(* Logix 5000 project; controller Google vendor 1 type 14 code 151 rev 31.11; software revision 31.00 *)

TASK MainTask (continuous, watchdog 500 ms) : MainProgram

MODULES
   Local : vendor 1 type 14 code 151 (Compact 0, rev 31.11)
      Discrete_IO : Embedded (Compact 1, rev 3.1, Output RPI 20 ms)
      Analog_IO : Embedded (Compact 2, rev 1.1, Output RPI 80 ms)
      Counters : Embedded (Compact 3, rev 1.1, Output RPI 20 ms)
      Lift_Main_Drive : PowerFlex 525-EENET (Ethernet 192.168.1.42, rev 5.1, Output RPI 50 ms)
      LST_1 : vendor 678 type 100 code 276 (Ethernet 192.168.1.149, rev 11.1, Output RPI 19 ms)
      LST_2 : vendor 678 type 100 code 276 (Ethernet 192.168.1.50, rev 11.1, Output RPI 17 ms)
      ToteCodeReader : vendor 678 type 773 code 1307 (Ethernet 192.168.1.151, rev 1.1, Output RPI 60 ms)
      L5_Conv : vendor 629 type 43 code 2 (Ethernet 192.168.1.165, rev 2.1, StandardDataDriven RPI 30 ms)
      L4_Conv : vendor 629 type 43 code 2 (Ethernet 192.168.1.164, rev 2.1, StandardDataDriven RPI 30 ms)
      L1_Conv : vendor 629 type 43 code 2 (Ethernet 192.168.1.161, rev 2.1, StandardDataDriven RPI 30 ms)
      Infeed_Conv : vendor 629 type 43 code 2 (Ethernet 192.168.1.160, rev 2.1, StandardDataDriven RPI 30 ms)
           Infeed_Conv:I.Data[0].0   // Zone 1 Sensor
           Infeed_Conv:I.Data[0].1   // Zone 2 Sensor
           Infeed_Conv:I.Data[0].2   // Zone 3 Sensor
           Infeed_Conv:I.Data[0].3   // Zone 4 Sensor
      L2_Conv : vendor 629 type 43 code 2 (Ethernet 192.168.1.162, rev 2.1, StandardDataDriven RPI 30 ms)
      L3_Conv : vendor 629 type 43 code 2 (Ethernet 192.168.1.163, rev 2.1, StandardDataDriven RPI 30 ms)
      Lift_Conv : vendor 629 type 43 code 2 (Ethernet 192.168.1.166, rev 2.1, StandardDataDriven RPI 30 ms)
END_MODULES

TYPE Addr :   // Structure UDT for MSG UDT
STRUCT
   Family : INT;   // 2 for IP4
   Port : INT;   // Remote Port Number
   Addr : DINT;   // Remote IP Address
END_STRUCT
END_TYPE

TYPE GIB_MSG :   // UDT Specified by Rockwell
STRUCT
   Instance : DINT;
   Addr : Addr;
END_STRUCT
END_TYPE

TYPE State :
STRUCT
   Stopped : DINT;
   Resetting : DINT;
   Ready : DINT;
   Starting : DINT;
   Running : DINT;
   Stopping : DINT;
END_STRUCT
END_TYPE

ADD_ON_INSTRUCTION Conv_Sensor_Inputs   (* revision 1.0 *)
VAR_INPUT
   Data : SINT; {required}
END_VAR
VAR_OUTPUT
   Input_0 : BOOL; {access Read Only, required}
   Input_1 : BOOL; {access Read Only, required}
   Input_2 : BOOL; {access Read Only, required}
   Input_3 : BOOL; {access Read Only, required}
END_VAR
VAR_INPUT
   Infeed_Mode : BOOL; {required}
   Outfeed_Mode : BOOL; {required}
   Outfeed_Stop_Delay : DINT; {required}
END_VAR
VAR
   Input_Delay : TIMER[4] := ([0].PRE := 1000, [1].PRE := 1000, [2].PRE := 1000, [3].PRE := 1000); {access None}
END_VAR

ROUTINE Logic   (* ladder *)
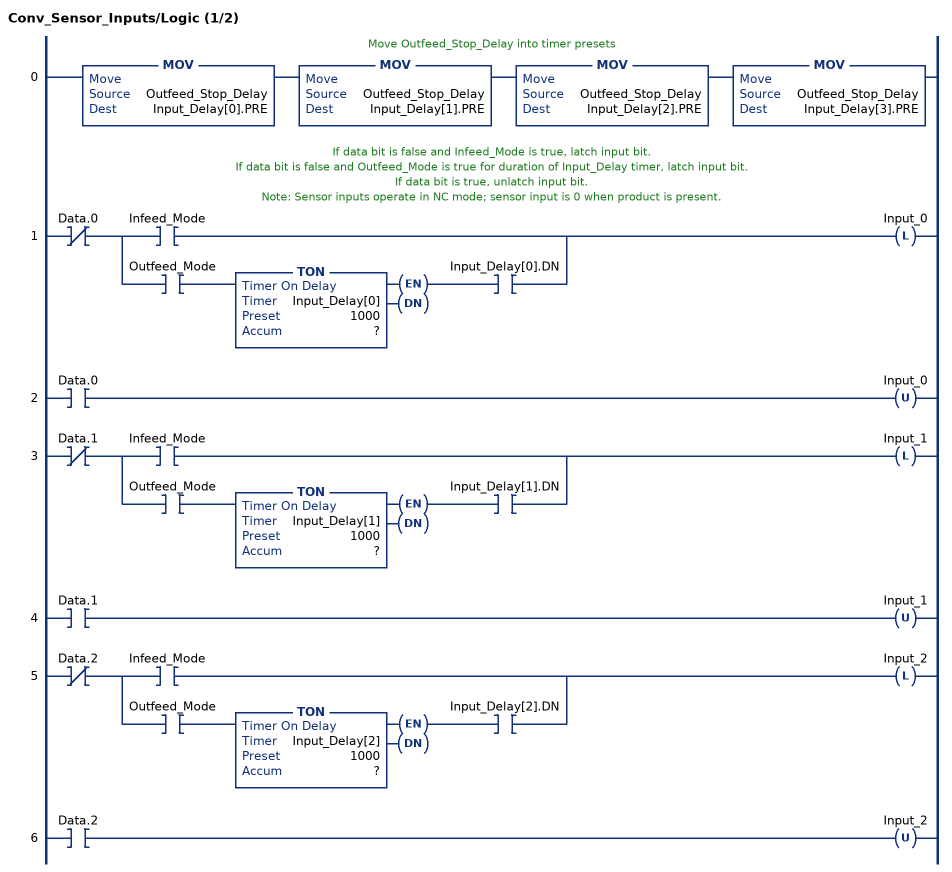
   // Move Outfeed_Stop_Delay into timer presets
   0: MOV(Outfeed_Stop_Delay,Input_Delay[0].PRE)MOV(Outfeed_Stop_Delay,Input_Delay[1].PRE)MOV(Outfeed_Stop_Delay,Input_Delay[2].PRE)MOV(Outfeed_Stop_Delay,Input_Delay[3].PRE);
   // If data bit is false and Infeed_Mode is true, latch input bit.
   // If data bit is false and Outfeed_Mode is true for duration of Input_Delay timer, latch input bit.
   // If data bit is true, unlatch input bit.
   // Note: Sensor inputs operate in NC mode; sensor input is 0 when product is present.
   1: XIO(Data.0)[XIC(Infeed_Mode) ,XIC(Outfeed_Mode) TON(Input_Delay[0],?,?) XIC(Input_Delay[0].DN) ]OTL(Input_0);
   2: XIC(Data.0)OTU(Input_0);
   3: XIO(Data.1)[XIC(Infeed_Mode) ,XIC(Outfeed_Mode) TON(Input_Delay[1],?,?) XIC(Input_Delay[1].DN) ]OTL(Input_1);
   4: XIC(Data.1)OTU(Input_1);
   5: XIO(Data.2)[XIC(Infeed_Mode) ,XIC(Outfeed_Mode) TON(Input_Delay[2],?,?) XIC(Input_Delay[2].DN) ]OTL(Input_2);
   6: XIC(Data.2)OTU(Input_2);
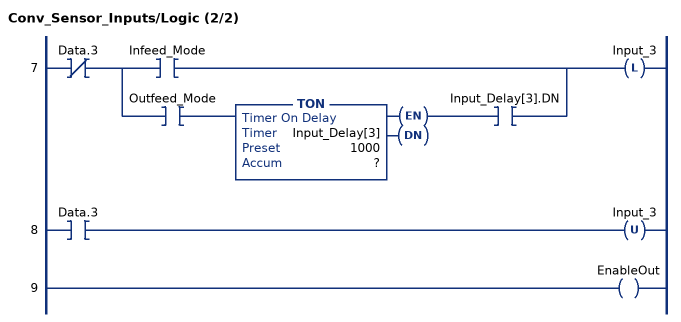
   7: XIO(Data.3)[XIC(Infeed_Mode) ,XIC(Outfeed_Mode) TON(Input_Delay[3],?,?) XIC(Input_Delay[3].DN) ]OTL(Input_3);
   8: XIC(Data.3)OTU(Input_3);
   9: OTE(EnableOut);
END_ROUTINE
END_ADD_ON_INSTRUCTION

ADD_ON_INSTRUCTION Conveyor_Motor_Control   (* revision 1.0 *)
VAR_OUTPUT
   Motor1_Data : SINT; {required}
   Motor2_Data : SINT; {access Read Only, required}
   Motor3_Data : SINT; {access Read Only, required}
   Motor4_Data : SINT; {access Read Only, required}
END_VAR
VAR_INPUT
   Motor1_FWD : BOOL; {required}
   Motor1_REV : BOOL; {required}
   Motor2_FWD : BOOL; {required}
   Motor2_REV : BOOL; {required}
   Motor3_FWD : BOOL; {required}
   Motor3_REV : BOOL; {required}
   Motor4_FWD : BOOL; {required}
   Motor4_REV : BOOL; {required}
   FWD_Speed : DINT; {required}
   REV_Speed : DINT; {required}
   Start_Delay : DINT; {required}
   Run_Permissive : DINT; {required}
END_VAR
VAR
   FWD_Delay : TIMER[4] := ([0].PRE := 500, [1].PRE := 500, [2].PRE := 500, [3].PRE := 500); {access None}
   REV_Delay : TIMER[4] := ([0].PRE := 500, [1].PRE := 500, [2].PRE := 500, [3].PRE := 500); {access None}
END_VAR

ROUTINE Logic   (* ladder *)
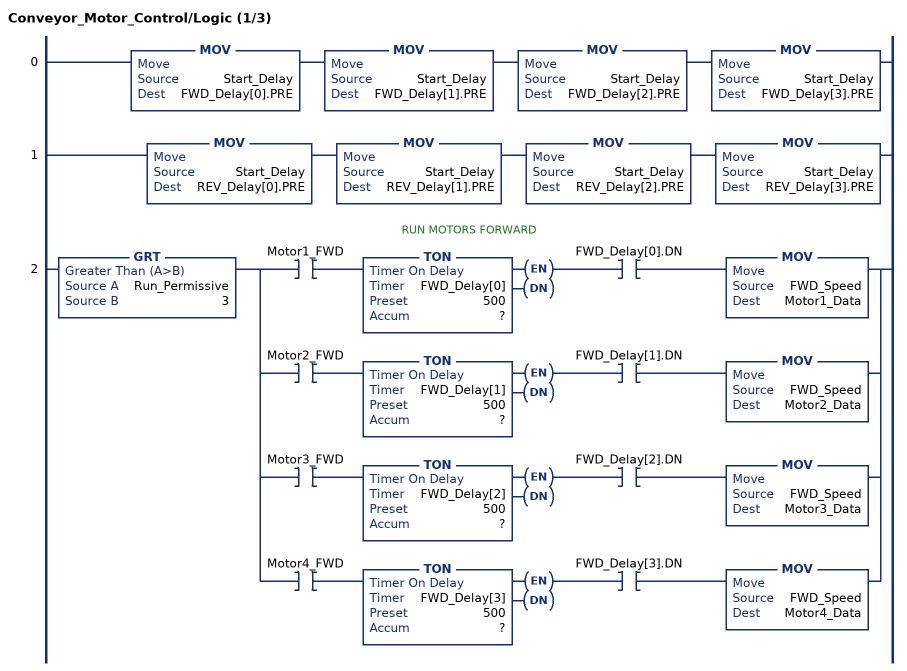
   0: MOV(Start_Delay,FWD_Delay[0].PRE)MOV(Start_Delay,FWD_Delay[1].PRE)MOV(Start_Delay,FWD_Delay[2].PRE)MOV(Start_Delay,FWD_Delay[3].PRE);
   1: MOV(Start_Delay,REV_Delay[0].PRE)MOV(Start_Delay,REV_Delay[1].PRE)MOV(Start_Delay,REV_Delay[2].PRE)MOV(Start_Delay,REV_Delay[3].PRE);
   // RUN MOTORS FORWARD
   2: GRT(Run_Permissive,3)[XIC(Motor1_FWD) TON(FWD_Delay[0],?,?) XIC(FWD_Delay[0].DN) MOV(FWD_Speed,Motor1_Data) ,XIC(Motor2_FWD) TON(FWD_Delay[1],?,?) XIC(FWD_Delay[1].DN) MOV(FWD_Speed,Motor2_Data) ,XIC(Motor3_FWD) TON(FWD_Delay[2],?,?) XIC(FWD_Delay[2].DN) MOV(FWD_Speed,Motor3_Data) ,XIC(Motor4_FWD) TON(FWD_Delay[3],?,?) XIC(FWD_Delay[3].DN) MOV(FWD_Speed,Motor4_Data) ];
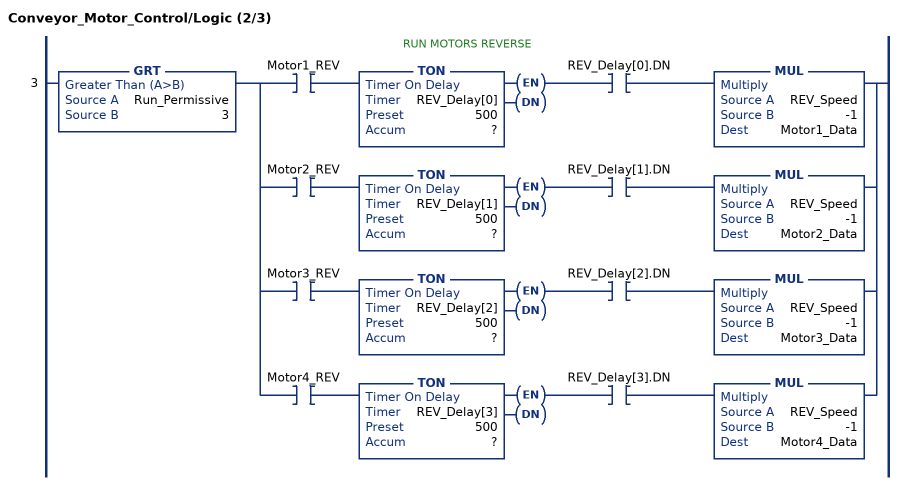
   // RUN MOTORS REVERSE
   3: GRT(Run_Permissive,3)[XIC(Motor1_REV) TON(REV_Delay[0],?,?) XIC(REV_Delay[0].DN) MUL(REV_Speed,-1,Motor1_Data) ,XIC(Motor2_REV) TON(REV_Delay[1],?,?) XIC(REV_Delay[1].DN) MUL(REV_Speed,-1,Motor2_Data) ,XIC(Motor3_REV) TON(REV_Delay[2],?,?) XIC(REV_Delay[2].DN) MUL(REV_Speed,-1,Motor3_Data) ,XIC(Motor4_REV) TON(REV_Delay[3],?,?) XIC(REV_Delay[3].DN) MUL(REV_Speed,-1,Motor4_Data) ];
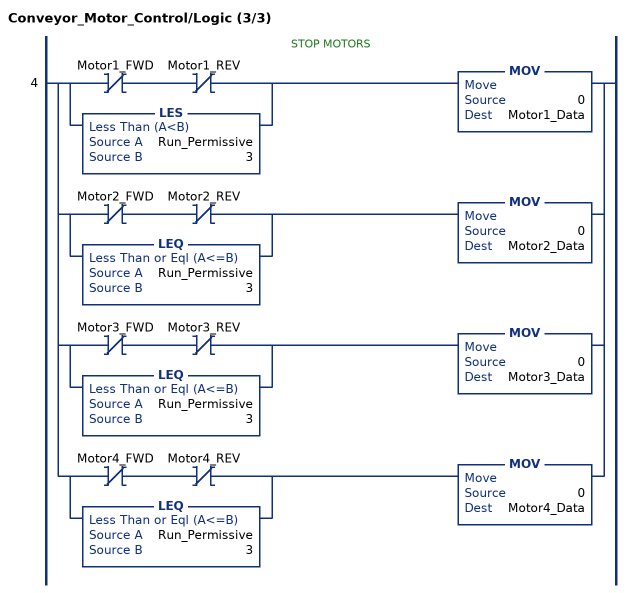
   // STOP MOTORS
   4: [[XIO(Motor1_FWD) XIO(Motor1_REV) ,LES(Run_Permissive,3) ] MOV(0,Motor1_Data) ,[XIO(Motor2_FWD) XIO(Motor2_REV) ,LEQ(Run_Permissive,3) ] MOV(0,Motor2_Data) ,[XIO(Motor3_FWD) XIO(Motor3_REV) ,LEQ(Run_Permissive,3) ] MOV(0,Motor3_Data) ,[XIO(Motor4_FWD) XIO(Motor4_REV) ,LEQ(Run_Permissive,3) ] MOV(0,Motor4_Data) ];
END_ROUTINE
END_ADD_ON_INSTRUCTION

ADD_ON_INSTRUCTION End_Zone_Data   (* revision 1.0 *)
VAR_IN_OUT
   Product_Name : STRING; {required}
   Product_Code : DINT; {required}
END_VAR
VAR_OUTPUT
   Occupied : BOOL; {access Read Only, visible}
END_VAR
VAR_INPUT
   Input : BOOL; {required}
END_VAR
VAR_IN_OUT
   Upstream_ProdName : STRING; {required}
   Upstream_ProdCode : DINT; {required}
END_VAR
VAR_INPUT
   FWD_Direction : BOOL; {required}
   REV_Direction : BOOL; {required}
END_VAR
VAR
   Blank_String : STRING; {access None}
   ONS : DINT; {access None}
   Occupied_Delay : TIMER := (PRE := 20); {access None}
END_VAR

ROUTINE Logic   (* ladder *)
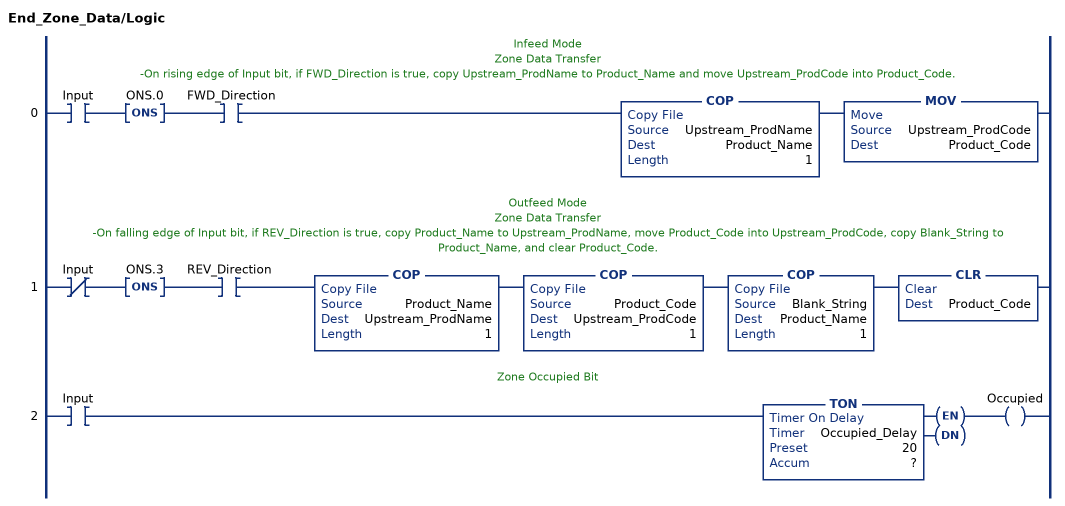
   // Infeed Mode
   // Zone Data Transfer
   // -On rising edge of Input bit, if FWD_Direction is true, copy Upstream_ProdName to Product_Name and move Upstream_ProdCode into Product_Code.
   0: XIC(Input)ONS(ONS.0)XIC(FWD_Direction)COP(Upstream_ProdName,Product_Name,1)MOV(Upstream_ProdCode,Product_Code);
   // Outfeed Mode
   // Zone Data Transfer
   // -On falling edge of Input bit, if REV_Direction is true, copy Product_Name to Upstream_ProdName, move Product_Code into Upstream_ProdCode, copy Blank_String to Product_Name, and clear Product_Code.
   1: XIO(Input)ONS(ONS.3)XIC(REV_Direction)COP(Product_Name,Upstream_ProdName,1)COP(Product_Code,Upstream_ProdCode,1)COP(Blank_String,Product_Name,1)CLR(Product_Code);
   // Zone Occupied Bit
   2: XIC(Input)TON(Occupied_Delay,?,?)OTE(Occupied);
END_ROUTINE
END_ADD_ON_INSTRUCTION

ADD_ON_INSTRUCTION Input_16_Bit   (* revision 1.0 *)
VAR_INPUT
   Data : INT; {required}
END_VAR
VAR_OUTPUT
   Input_0 : BOOL; {access Read Only, required}
END_VAR
VAR_INPUT
   Input0_On_Debounce : DINT; {required}
   Input0_Off_Debounce : DINT; {required}
END_VAR
VAR_OUTPUT
   Input_1 : BOOL; {access Read Only, required}
END_VAR
VAR_INPUT
   Input1_On_Debounce : DINT; {required}
   Input1_Off_Debounce : DINT; {required}
END_VAR
VAR_OUTPUT
   Input_2 : BOOL; {access Read Only, required}
END_VAR
VAR_INPUT
   Input2_On_Debounce : DINT; {required}
   Input2_Off_Debounce : DINT; {required}
END_VAR
VAR_OUTPUT
   Input_3 : BOOL; {access Read Only, required}
END_VAR
VAR_INPUT
   Input3_On_Debounce : DINT; {required}
   Input3_Off_Debounce : DINT; {required}
END_VAR
VAR_OUTPUT
   Input_4 : BOOL; {access Read Only, required}
END_VAR
VAR_INPUT
   Input4_On_Debounce : DINT; {required}
   Input4_Off_Debounce : DINT; {required}
END_VAR
VAR_OUTPUT
   Input_5 : BOOL; {access Read Only, required}
END_VAR
VAR_INPUT
   Input5_On_Debounce : DINT; {required}
   Input5_Off_Debounce : DINT; {required}
END_VAR
VAR_OUTPUT
   Input_6 : BOOL; {access Read Only, required}
END_VAR
VAR_INPUT
   Input6_On_Debounce : DINT; {required}
   Input6_Off_Debounce : DINT; {required}
END_VAR
VAR_OUTPUT
   Input_7 : BOOL; {access Read Only, required}
END_VAR
VAR_INPUT
   Input7_On_Debounce : DINT; {required}
   Input7_Off_Debounce : DINT; {required}
END_VAR
VAR_OUTPUT
   Input_8 : BOOL; {access Read Only, required}
END_VAR
VAR_INPUT
   Input8_On_Debounce : DINT; {required}
   Input8_Off_Debounce : DINT; {required}
END_VAR
VAR_OUTPUT
   Input_9 : BOOL; {access Read Only, required}
END_VAR
VAR_INPUT
   Input9_On_Debounce : DINT; {required}
   Input9_Off_Debounce : DINT; {required}
END_VAR
VAR_OUTPUT
   Input_10 : BOOL; {access Read Only, required}
END_VAR
VAR_INPUT
   Input10_On_Debounce : DINT; {required}
   Input10_Off_Debounce : DINT; {required}
END_VAR
VAR_OUTPUT
   Input_11 : BOOL; {access Read Only, required}
END_VAR
VAR_INPUT
   Input11_On_Debounce : DINT; {required}
   Input11_Off_Debounce : DINT; {required}
END_VAR
VAR_OUTPUT
   Input_12 : BOOL; {access Read Only, required}
END_VAR
VAR_INPUT
   Input12_On_Debounce : DINT; {required}
   Input12_Off_Debounce : DINT; {required}
END_VAR
VAR_OUTPUT
   Input_13 : BOOL; {access Read Only, required}
END_VAR
VAR_INPUT
   Input13_On_Debounce : DINT; {required}
   Input13_Off_Debounce : DINT; {required}
END_VAR
VAR_OUTPUT
   Input_14 : BOOL; {access Read Only, required}
END_VAR
VAR_INPUT
   Input14_On_Debounce : DINT; {required}
   Input14_Off_Debounce : DINT; {required}
END_VAR
VAR_OUTPUT
   Input_15 : BOOL; {access Read Only, required}
END_VAR
VAR_INPUT
   Input15_On_Debounce : DINT; {required}
   Input15_Off_Debounce : DINT; {required}
END_VAR
VAR
   Debounce_On_TMR : TIMER[16]; {access None}
   Debounce_Off_TMR : TIMER[16]; {access None}
END_VAR

ROUTINE Logic   (* ladder *)
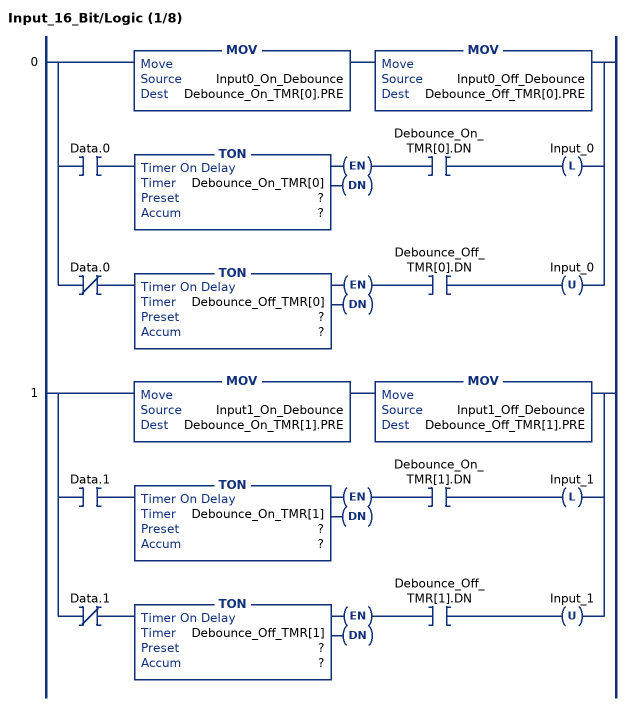
   0: [MOV(Input0_On_Debounce,Debounce_On_TMR[0].PRE) MOV(Input0_Off_Debounce,Debounce_Off_TMR[0].PRE) ,[XIC(Data.0) TON(Debounce_On_TMR[0],?,?) XIC(Debounce_On_TMR[0].DN) OTL(Input_0) ,XIO(Data.0) TON(Debounce_Off_TMR[0],?,?) XIC(Debounce_Off_TMR[0].DN) OTU(Input_0) ] ];
   1: [MOV(Input1_On_Debounce,Debounce_On_TMR[1].PRE) MOV(Input1_Off_Debounce,Debounce_Off_TMR[1].PRE) ,[XIC(Data.1) TON(Debounce_On_TMR[1],?,?) XIC(Debounce_On_TMR[1].DN) OTL(Input_1) ,XIO(Data.1) TON(Debounce_Off_TMR[1],?,?) XIC(Debounce_Off_TMR[1].DN) OTU(Input_1) ] ];
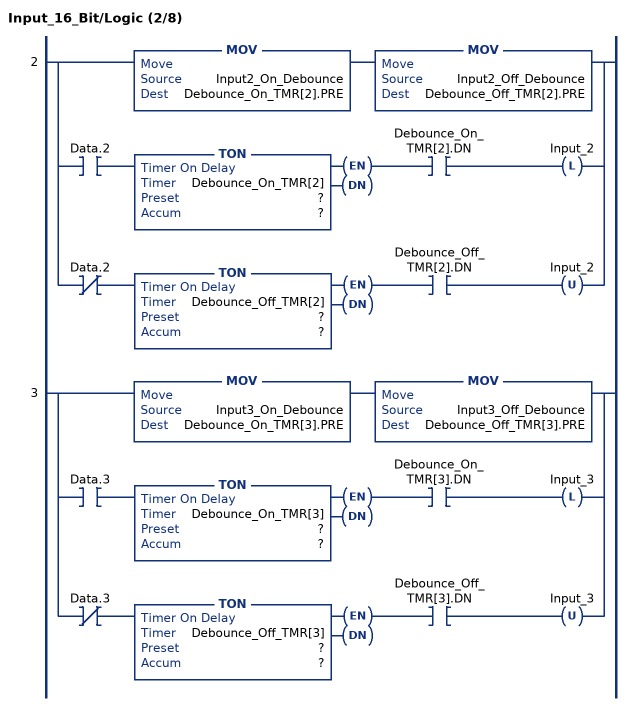
   2: [MOV(Input2_On_Debounce,Debounce_On_TMR[2].PRE) MOV(Input2_Off_Debounce,Debounce_Off_TMR[2].PRE) ,[XIC(Data.2) TON(Debounce_On_TMR[2],?,?) XIC(Debounce_On_TMR[2].DN) OTL(Input_2) ,XIO(Data.2) TON(Debounce_Off_TMR[2],?,?) XIC(Debounce_Off_TMR[2].DN) OTU(Input_2) ] ];
   3: [MOV(Input3_On_Debounce,Debounce_On_TMR[3].PRE) MOV(Input3_Off_Debounce,Debounce_Off_TMR[3].PRE) ,[XIC(Data.3) TON(Debounce_On_TMR[3],?,?) XIC(Debounce_On_TMR[3].DN) OTL(Input_3) ,XIO(Data.3) TON(Debounce_Off_TMR[3],?,?) XIC(Debounce_Off_TMR[3].DN) OTU(Input_3) ] ];
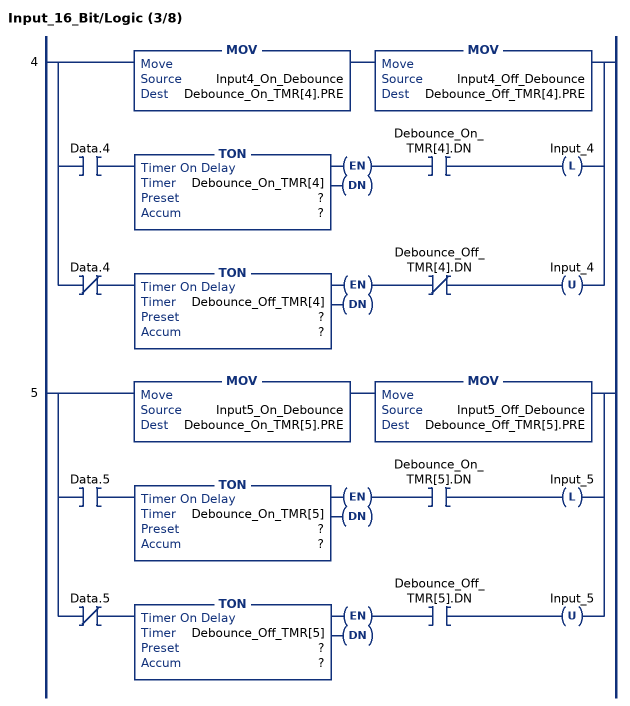
   4: [MOV(Input4_On_Debounce,Debounce_On_TMR[4].PRE) MOV(Input4_Off_Debounce,Debounce_Off_TMR[4].PRE) ,[XIC(Data.4) TON(Debounce_On_TMR[4],?,?) XIC(Debounce_On_TMR[4].DN) OTL(Input_4) ,XIO(Data.4) TON(Debounce_Off_TMR[4],?,?) XIO(Debounce_Off_TMR[4].DN) OTU(Input_4) ] ];
   5: [MOV(Input5_On_Debounce,Debounce_On_TMR[5].PRE) MOV(Input5_Off_Debounce,Debounce_Off_TMR[5].PRE) ,[XIC(Data.5) TON(Debounce_On_TMR[5],?,?) XIC(Debounce_On_TMR[5].DN) OTL(Input_5) ,XIO(Data.5) TON(Debounce_Off_TMR[5],?,?) XIC(Debounce_Off_TMR[5].DN) OTU(Input_5) ] ];
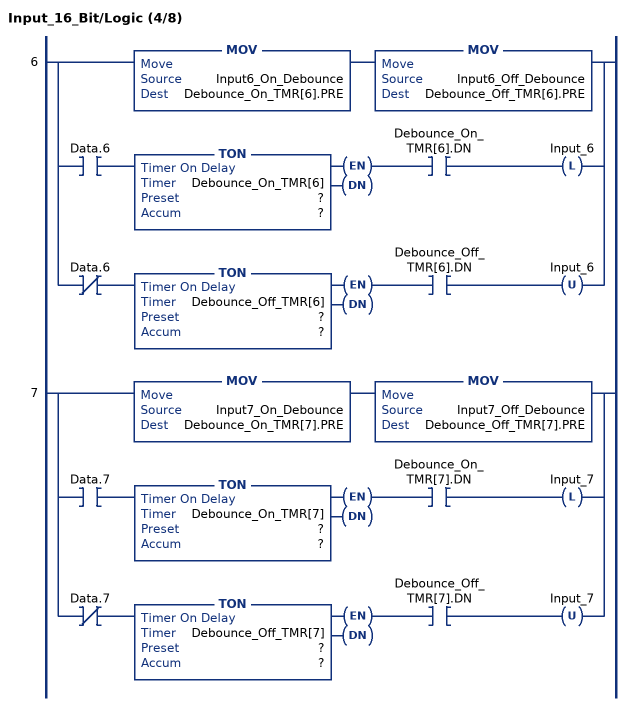
   6: [MOV(Input6_On_Debounce,Debounce_On_TMR[6].PRE) MOV(Input6_Off_Debounce,Debounce_Off_TMR[6].PRE) ,[XIC(Data.6) TON(Debounce_On_TMR[6],?,?) XIC(Debounce_On_TMR[6].DN) OTL(Input_6) ,XIO(Data.6) TON(Debounce_Off_TMR[6],?,?) XIC(Debounce_Off_TMR[6].DN) OTU(Input_6) ] ];
   7: [MOV(Input7_On_Debounce,Debounce_On_TMR[7].PRE) MOV(Input7_Off_Debounce,Debounce_Off_TMR[7].PRE) ,[XIC(Data.7) TON(Debounce_On_TMR[7],?,?) XIC(Debounce_On_TMR[7].DN) OTL(Input_7) ,XIO(Data.7) TON(Debounce_Off_TMR[7],?,?) XIC(Debounce_Off_TMR[7].DN) OTU(Input_7) ] ];
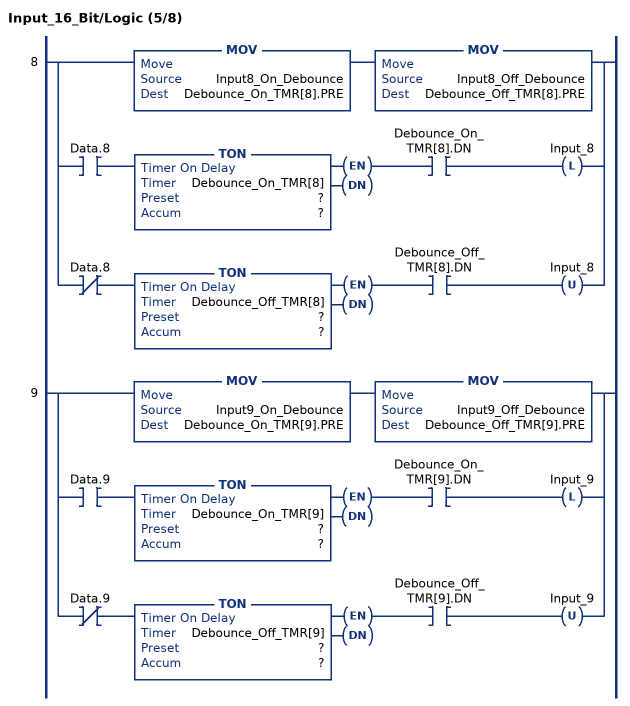
   8: [MOV(Input8_On_Debounce,Debounce_On_TMR[8].PRE) MOV(Input8_Off_Debounce,Debounce_Off_TMR[8].PRE) ,[XIC(Data.8) TON(Debounce_On_TMR[8],?,?) XIC(Debounce_On_TMR[8].DN) OTL(Input_8) ,XIO(Data.8) TON(Debounce_Off_TMR[8],?,?) XIC(Debounce_Off_TMR[8].DN) OTU(Input_8) ] ];
   9: [MOV(Input9_On_Debounce,Debounce_On_TMR[9].PRE) MOV(Input9_Off_Debounce,Debounce_Off_TMR[9].PRE) ,[XIC(Data.9) TON(Debounce_On_TMR[9],?,?) XIC(Debounce_On_TMR[9].DN) OTL(Input_9) ,XIO(Data.9) TON(Debounce_Off_TMR[9],?,?) XIC(Debounce_Off_TMR[9].DN) OTU(Input_9) ] ];
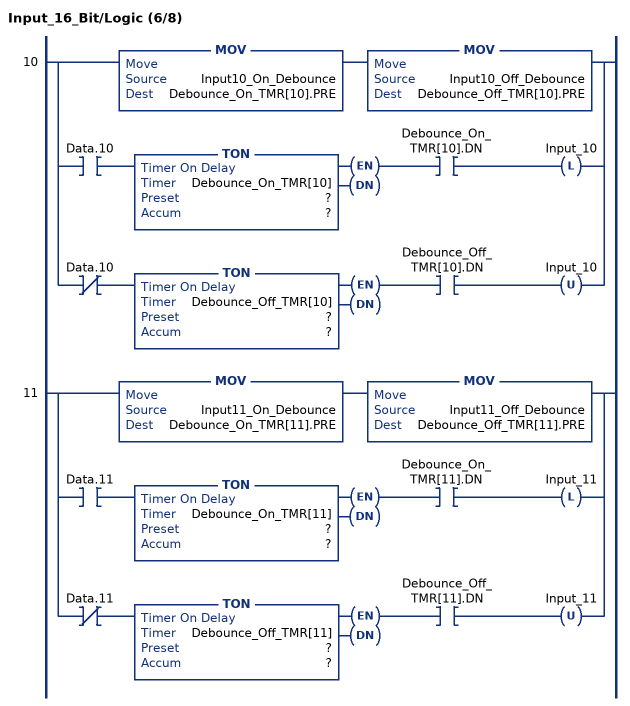
   10: [MOV(Input10_On_Debounce,Debounce_On_TMR[10].PRE) MOV(Input10_Off_Debounce,Debounce_Off_TMR[10].PRE) ,[XIC(Data.10) TON(Debounce_On_TMR[10],?,?) XIC(Debounce_On_TMR[10].DN) OTL(Input_10) ,XIO(Data.10) TON(Debounce_Off_TMR[10],?,?) XIC(Debounce_Off_TMR[10].DN) OTU(Input_10) ] ];
   11: [MOV(Input11_On_Debounce,Debounce_On_TMR[11].PRE) MOV(Input11_Off_Debounce,Debounce_Off_TMR[11].PRE) ,[XIC(Data.11) TON(Debounce_On_TMR[11],?,?) XIC(Debounce_On_TMR[11].DN) OTL(Input_11) ,XIO(Data.11) TON(Debounce_Off_TMR[11],?,?) XIC(Debounce_Off_TMR[11].DN) OTU(Input_11) ] ];
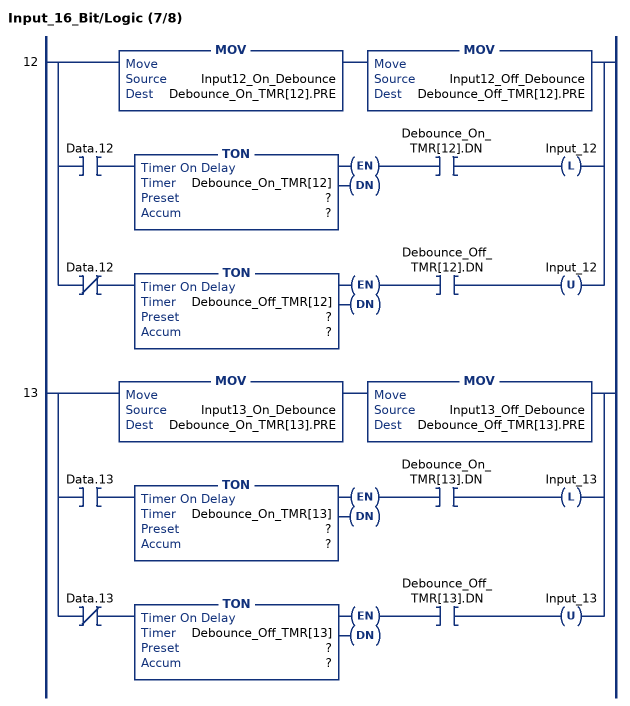
   12: [MOV(Input12_On_Debounce,Debounce_On_TMR[12].PRE) MOV(Input12_Off_Debounce,Debounce_Off_TMR[12].PRE) ,[XIC(Data.12) TON(Debounce_On_TMR[12],?,?) XIC(Debounce_On_TMR[12].DN) OTL(Input_12) ,XIO(Data.12) TON(Debounce_Off_TMR[12],?,?) XIC(Debounce_Off_TMR[12].DN) OTU(Input_12) ] ];
   13: [MOV(Input13_On_Debounce,Debounce_On_TMR[13].PRE) MOV(Input13_Off_Debounce,Debounce_Off_TMR[13].PRE) ,[XIC(Data.13) TON(Debounce_On_TMR[13],?,?) XIC(Debounce_On_TMR[13].DN) OTL(Input_13) ,XIO(Data.13) TON(Debounce_Off_TMR[13],?,?) XIC(Debounce_Off_TMR[13].DN) OTU(Input_13) ] ];
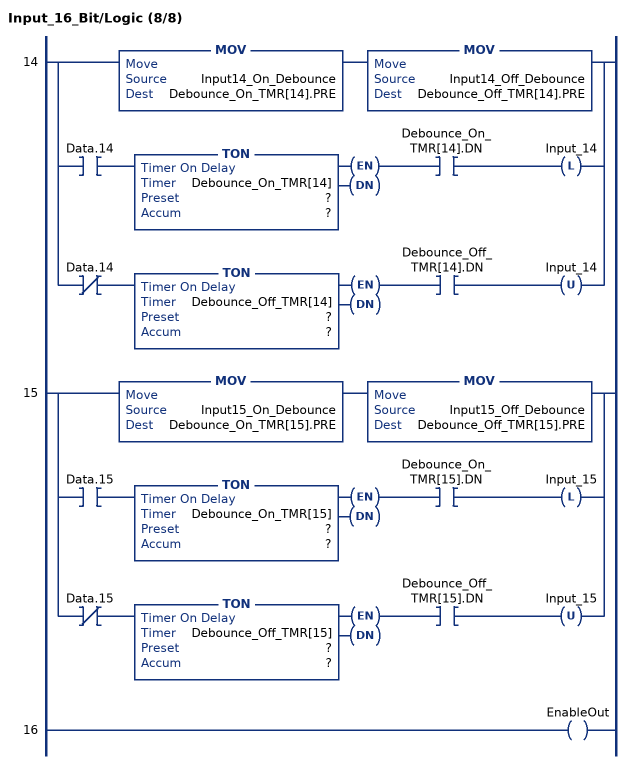
   14: [MOV(Input14_On_Debounce,Debounce_On_TMR[14].PRE) MOV(Input14_Off_Debounce,Debounce_Off_TMR[14].PRE) ,[XIC(Data.14) TON(Debounce_On_TMR[14],?,?) XIC(Debounce_On_TMR[14].DN) OTL(Input_14) ,XIO(Data.14) TON(Debounce_Off_TMR[14],?,?) XIC(Debounce_Off_TMR[14].DN) OTU(Input_14) ] ];
   15: [MOV(Input15_On_Debounce,Debounce_On_TMR[15].PRE) MOV(Input15_Off_Debounce,Debounce_Off_TMR[15].PRE) ,[XIC(Data.15) TON(Debounce_On_TMR[15],?,?) XIC(Debounce_On_TMR[15].DN) OTL(Input_15) ,XIO(Data.15) TON(Debounce_Off_TMR[15],?,?) XIC(Debounce_Off_TMR[15].DN) OTU(Input_15) ] ];
   16: OTE(EnableOut);
END_ROUTINE
END_ADD_ON_INSTRUCTION

ADD_ON_INSTRUCTION Input_8_Bit   (* revision 1.0 *)
VAR_INPUT
   Data : SINT; {required}
END_VAR
VAR_OUTPUT
   Input_0 : BOOL; {access Read Only, required}
END_VAR
VAR_INPUT
   Input0_On_Debounce : DINT; {required}
   Input0_Off_Debounce : DINT; {required}
END_VAR
VAR_OUTPUT
   Input_1 : BOOL; {access Read Only, required}
END_VAR
VAR_INPUT
   Input1_On_Debounce : DINT; {required}
   Input1_Off_Debounce : DINT; {required}
END_VAR
VAR_OUTPUT
   Input_2 : BOOL; {access Read Only, required}
END_VAR
VAR_INPUT
   Input2_On_Debounce : DINT; {required}
   Input2_Off_Debounce : DINT; {required}
END_VAR
VAR_OUTPUT
   Input_3 : BOOL; {access Read Only, required}
END_VAR
VAR_INPUT
   Input3_On_Debounce : DINT; {required}
   Input3_Off_Debounce : DINT; {required}
END_VAR
VAR_OUTPUT
   Input_4 : BOOL; {access Read Only, required}
END_VAR
VAR_INPUT
   Input4_On_Debounce : DINT; {required}
   Input4_Off_Debounce : DINT; {required}
END_VAR
VAR_OUTPUT
   Input_5 : BOOL; {access Read Only, required}
END_VAR
VAR_INPUT
   Input5_On_Debounce : DINT; {required}
   Input5_Off_Debounce : DINT; {required}
END_VAR
VAR_OUTPUT
   Input_6 : BOOL; {access Read Only, required}
END_VAR
VAR_INPUT
   Input6_On_Debounce : DINT; {required}
   Input6_Off_Debounce : DINT; {required}
END_VAR
VAR_OUTPUT
   Input_7 : BOOL; {access Read Only, required}
END_VAR
VAR_INPUT
   Input7_On_Debounce : DINT; {required}
   Input7_Off_Debounce : DINT; {required}
END_VAR
VAR
   Debounce_On_TMR : TIMER[16]; {access None}
   Debounce_Off_TMR : TIMER[16]; {access None}
END_VAR

ROUTINE Logic   (* ladder *)
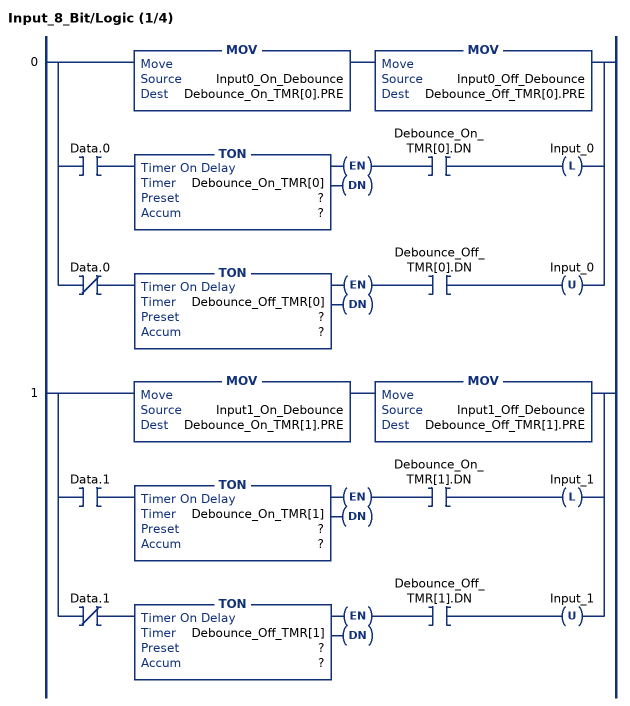
   0: [MOV(Input0_On_Debounce,Debounce_On_TMR[0].PRE) MOV(Input0_Off_Debounce,Debounce_Off_TMR[0].PRE) ,[XIC(Data.0) TON(Debounce_On_TMR[0],?,?) XIC(Debounce_On_TMR[0].DN) OTL(Input_0) ,XIO(Data.0) TON(Debounce_Off_TMR[0],?,?) XIC(Debounce_Off_TMR[0].DN) OTU(Input_0) ] ];
   1: [MOV(Input1_On_Debounce,Debounce_On_TMR[1].PRE) MOV(Input1_Off_Debounce,Debounce_Off_TMR[1].PRE) ,[XIC(Data.1) TON(Debounce_On_TMR[1],?,?) XIC(Debounce_On_TMR[1].DN) OTL(Input_1) ,XIO(Data.1) TON(Debounce_Off_TMR[1],?,?) XIC(Debounce_Off_TMR[1].DN) OTU(Input_1) ] ];
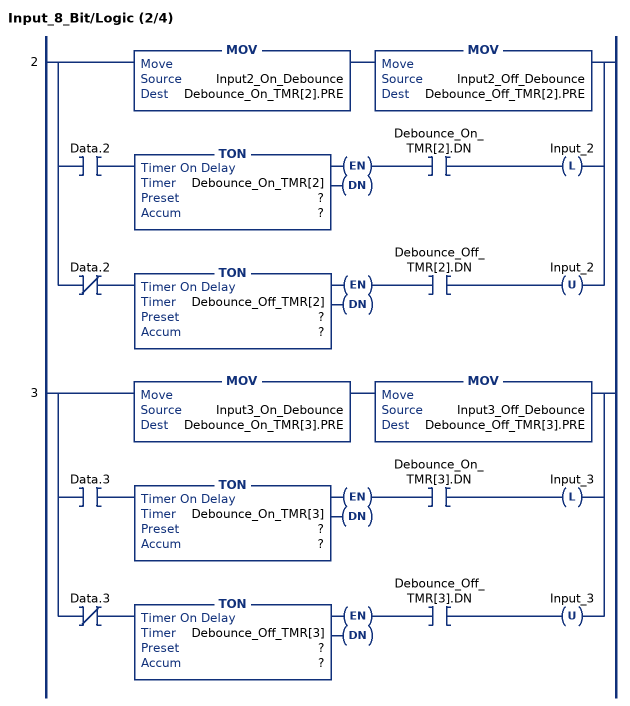
   2: [MOV(Input2_On_Debounce,Debounce_On_TMR[2].PRE) MOV(Input2_Off_Debounce,Debounce_Off_TMR[2].PRE) ,[XIC(Data.2) TON(Debounce_On_TMR[2],?,?) XIC(Debounce_On_TMR[2].DN) OTL(Input_2) ,XIO(Data.2) TON(Debounce_Off_TMR[2],?,?) XIC(Debounce_Off_TMR[2].DN) OTU(Input_2) ] ];
   3: [MOV(Input3_On_Debounce,Debounce_On_TMR[3].PRE) MOV(Input3_Off_Debounce,Debounce_Off_TMR[3].PRE) ,[XIC(Data.3) TON(Debounce_On_TMR[3],?,?) XIC(Debounce_On_TMR[3].DN) OTL(Input_3) ,XIO(Data.3) TON(Debounce_Off_TMR[3],?,?) XIC(Debounce_Off_TMR[3].DN) OTU(Input_3) ] ];
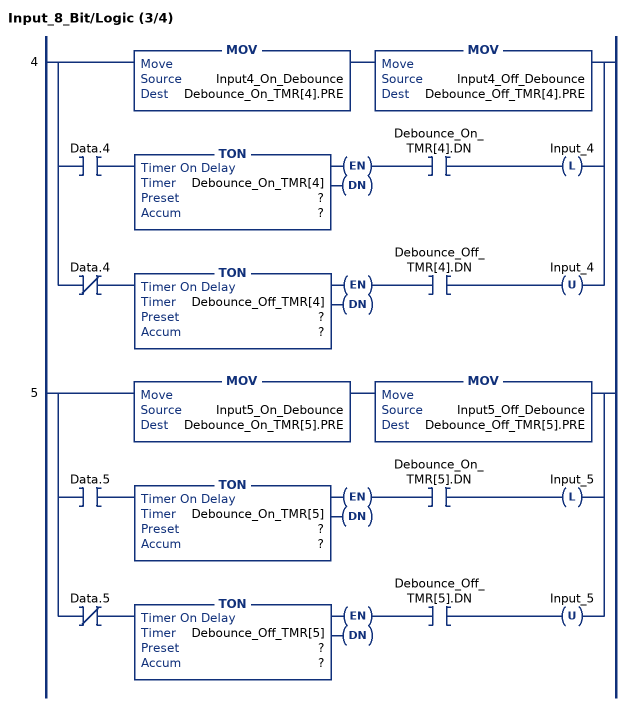
   4: [MOV(Input4_On_Debounce,Debounce_On_TMR[4].PRE) MOV(Input4_Off_Debounce,Debounce_Off_TMR[4].PRE) ,[XIC(Data.4) TON(Debounce_On_TMR[4],?,?) XIC(Debounce_On_TMR[4].DN) OTL(Input_4) ,XIO(Data.4) TON(Debounce_Off_TMR[4],?,?) XIC(Debounce_Off_TMR[4].DN) OTU(Input_4) ] ];
   5: [MOV(Input5_On_Debounce,Debounce_On_TMR[5].PRE) MOV(Input5_Off_Debounce,Debounce_Off_TMR[5].PRE) ,[XIC(Data.5) TON(Debounce_On_TMR[5],?,?) XIC(Debounce_On_TMR[5].DN) OTL(Input_5) ,XIO(Data.5) TON(Debounce_Off_TMR[5],?,?) XIC(Debounce_Off_TMR[5].DN) OTU(Input_5) ] ];
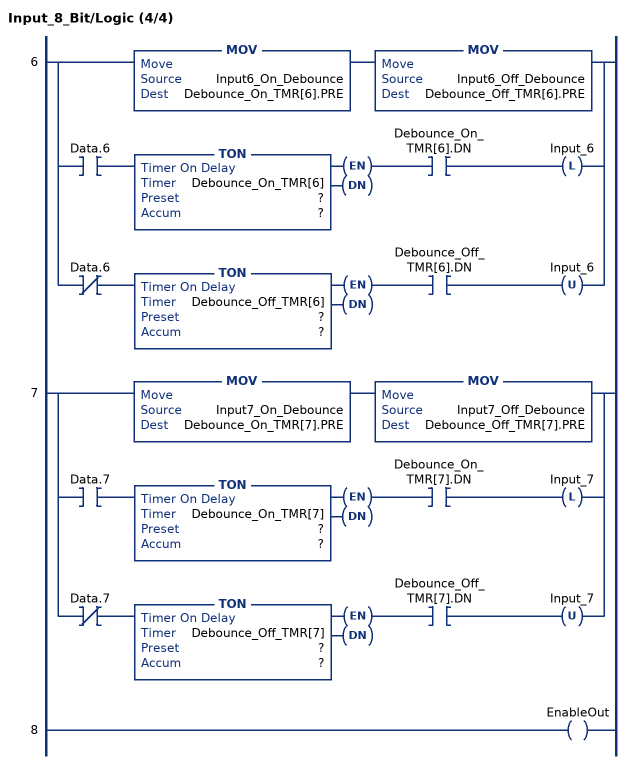
   6: [MOV(Input6_On_Debounce,Debounce_On_TMR[6].PRE) MOV(Input6_Off_Debounce,Debounce_Off_TMR[6].PRE) ,[XIC(Data.6) TON(Debounce_On_TMR[6],?,?) XIC(Debounce_On_TMR[6].DN) OTL(Input_6) ,XIO(Data.6) TON(Debounce_Off_TMR[6],?,?) XIC(Debounce_Off_TMR[6].DN) OTU(Input_6) ] ];
   7: [MOV(Input7_On_Debounce,Debounce_On_TMR[7].PRE) MOV(Input7_Off_Debounce,Debounce_Off_TMR[7].PRE) ,[XIC(Data.7) TON(Debounce_On_TMR[7],?,?) XIC(Debounce_On_TMR[7].DN) OTL(Input_7) ,XIO(Data.7) TON(Debounce_Off_TMR[7],?,?) XIC(Debounce_Off_TMR[7].DN) OTU(Input_7) ] ];
   8: OTE(EnableOut);
END_ROUTINE
END_ADD_ON_INSTRUCTION
